FUNCTION_BLOCK PUBLIC StartCommand EXTENDS CommandBase
VAR_INPUT
END_VAR
VAR_OUTPUT	
	Q : BOOL;
END_VAR
VAR
END_VAR

METHOD PROTECTED Task : BOOL
VAR_INPUT
	Init 	: BOOL;		// True the first time the Task is called after Execute is started
END_VAR
IF (NOT Init AND Q) THEN
	// Task comlete;
	Task := SUPER^.Task(Init);;
END_IF

// set init
Q := Init;
END_METHOD

END_FUNCTION_BLOCK

(* stored: Version 1.1.0.1, ProductVersion 3.1.4022.10
   POU StartCommand: Id {1855cea0-8f60-01cb-2735-aec5fa1a116a}, SpecialFunc None
   Method Task: Id {31cbc226-8269-0d51-3e95-0f735a54ab0d} *)
